(* Schneider Machine Expert - Basic project 152024, file version 2.7.0.0 *)
(* ProjectInformations: Name=New project *)

HARDWARE
  Cpu 0: TM221CE16R
  ModuleExtensionObject 0: TM3DM24R/G
  EthernetConfiguration: NetworkName=M221, IpAllocationMode=FixedAddress, IpAddress=0.0.0.0, SubnetMask=0.0.0.0
  SerialLineConfiguration: Baud=Baud19200, Parity=ParityEven, DataBits=DataBits8, StopBits=StopBits1, PhysicalMedium=PhysicalMediumRs485, TransmissionMode=TransmissionModeModbusRtu, SlaveId=1, Addressing=SlaveAddressing
  MastTask: UsePeriodScanMode=false, PeriodScan=100
  FastTask: Period=255
  CpuBehavior: StartingMode=StartAsPreviousState, AutoSaveRamOnEeprom=true, WatchdogPeriod=250

SYMBOLS  (address, symbol, comment, settings)
  %M0       WATF4  "Was At Floor 4"
  %M1       WATF1  "Was At Floor 1"
  %M2       WATF2  "Was At Floor 2"
  %M3       WATF3  "Was At Floor 3"
  %M4       F1CALL
  %M5       F2CALL
  %M6       F3CALL
  %M7       ATF1  "At Floor 1"
  %M8       ATF2  "At Floor 2"
  %M9       ATF3  "At Floor 3"
  %M10      F4CALL
  %M11      ATF4
  %M12      DOOR_CNT
  %M30      F1LATCH
  %M31      F2LATCH
  %M32      F3LATCH
  %M35        "attaxk"
  %TM0        [Preset=5000, Base=OneMilliSeconds]
  %TM1        [Preset=1000, Base=OneMilliSeconds]
  %TM2        [Preset=30]
  %TM3        [Preset=7, Base=OneSecond]
  %I0.0     LS1
  %I0.1     LS2
  %I0.2     LS3
  %I0.3     LDR_CLOSE
  %I0.4     ECB4
  %I0.5     ECB1
  %I0.6     ECB2
  %I0.7     ECB3
  %I0.8     LDR_OPEN
  %Q0.0     UP
  %Q0.1     DOWN
  %Q0.2     FD_C
  %Q0.3     DOOR_OPEN
  %Q0.4     FD_AGD
  %Q0.5     FD_E
  %Q0.6     FD_CLOSE

POU What Floor
  (* SectionNumber=0 *)

// Rung 0
  LD %I0.0                (* LS1 *)
  S %M1                   (* WATF1 *)
  R %M2                   (* WATF2 *)
  R %M3                   (* WATF3 *)
  ST %M7                  (* ATF1 *)
  R %M0                   (* WATF4 *)
  // as ST:
  //   IF LS1 THEN WATF1 := TRUE; END_IF;
  //   IF LS1 THEN WATF2 := FALSE; END_IF;
  //   IF LS1 THEN WATF3 := FALSE; END_IF;
  //   ATF1 := LS1;
  //   IF LS1 THEN WATF4 := FALSE; END_IF;

// Rung 1
  LD %I0.1                (* LS2 *)
  R %M1                   (* WATF1 *)
  S %M2                   (* WATF2 *)
  R %M3                   (* WATF3 *)
  ST %M8                  (* ATF2 *)
  R %M0                   (* WATF4 *)
  // as ST:
  //   IF LS2 THEN WATF1 := FALSE; END_IF;
  //   IF LS2 THEN WATF2 := TRUE; END_IF;
  //   IF LS2 THEN WATF3 := FALSE; END_IF;
  //   ATF2 := LS2;
  //   IF LS2 THEN WATF4 := FALSE; END_IF;

// Rung 2
  LD %I0.2                (* LS3 *)
  R %M1                   (* WATF1 *)
  R %M2                   (* WATF2 *)
  S %M3                   (* WATF3 *)
  ST %M9                  (* ATF3 *)
  R %M0                   (* WATF4 *)
  // as ST:
  //   IF LS3 THEN WATF1 := FALSE; END_IF;
  //   IF LS3 THEN WATF2 := FALSE; END_IF;
  //   IF LS3 THEN WATF3 := TRUE; END_IF;
  //   ATF3 := LS3;
  //   IF LS3 THEN WATF4 := FALSE; END_IF;

POU First Called
  (* SectionNumber=0 *)

// Rung 3
  LD %I0.5                (* ECB1 *)
  ANDN %M7                (* ATF1 *)
  S %M4                   (* F1CALL *)
  // as ST:
  //   IF ECB1 AND NOT ATF1 THEN F1CALL := TRUE; END_IF;

// Rung 4
  LD %M4                  (* F1CALL *)
  S %Q0.1                 (* DOWN *)
  // as ST:
  //   IF F1CALL THEN DOWN := TRUE; END_IF;

// Rung 5
  LD %M7                  (* ATF1 *)
  AND %M4                 (* F1CALL *)
  R %Q0.1                 (* DOWN *)
  // as ST:
  //   IF ATF1 AND F1CALL THEN DOWN := FALSE; END_IF;

// Rung 6
  LD %M7                  (* ATF1 *)
  R %M4                   (* F1CALL *)
  // as ST:
  //   IF ATF1 THEN F1CALL := FALSE; END_IF;

POU Second Called
  (* SectionNumber=0 *)

// Rung 7
  LD %I0.6                (* ECB2 *)
  ANDN %M8                (* ATF2 *)
  S %M5                   (* F2CALL *)
  // as ST:
  //   IF ECB2 AND NOT ATF2 THEN F2CALL := TRUE; END_IF;

// Rung 8
  LD %M5                  (* F2CALL *)
  AND %M1                 (* WATF1 *)
  S %Q0.0                 (* UP *)
  // as ST:
  //   IF F2CALL AND WATF1 THEN UP := TRUE; END_IF;

// Rung 9
  LD %M5                  (* F2CALL *)
  AND( %M3                (* WATF3 *)
  OR %M0                  (* WATF4 *)
  )
  S %Q0.1                 (* DOWN *)
  // as ST:
  //   IF F2CALL AND (WATF3 OR WATF4) THEN DOWN := TRUE; END_IF;

// Rung 10
  LD %M8                  (* ATF2 *)
  AND %M5                 (* F2CALL *)
  R %Q0.0                 (* UP *)
  R %Q0.1                 (* DOWN *)
  // as ST:
  //   IF ATF2 AND F2CALL THEN UP := FALSE; END_IF;
  //   IF ATF2 AND F2CALL THEN DOWN := FALSE; END_IF;

// Rung 11
  LD %M8                  (* ATF2 *)
  R %M5                   (* F2CALL *)
  // as ST:
  //   IF ATF2 THEN F2CALL := FALSE; END_IF;

POU Third Called
  (* SectionNumber=0 *)

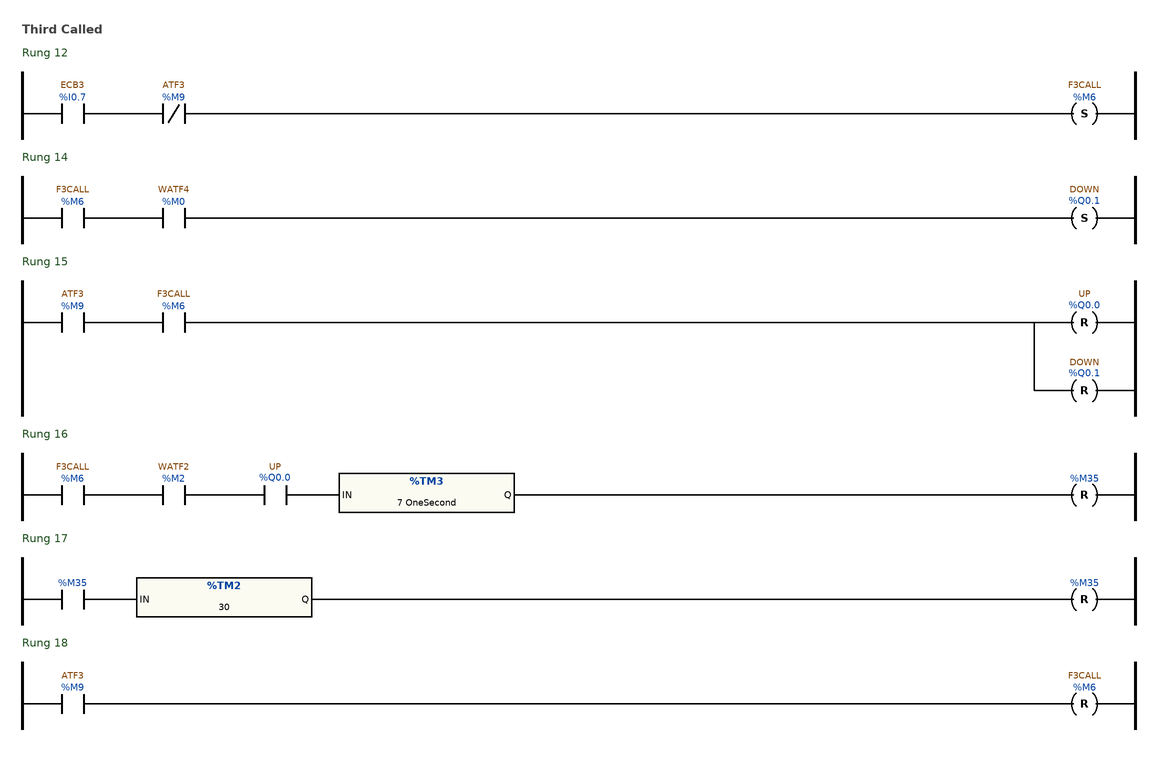

// Rung 12
  LD %I0.7                (* ECB3 *)
  ANDN %M9                (* ATF3 *)
  S %M6                   (* F3CALL *)
  // as ST:
  //   IF ECB3 AND NOT ATF3 THEN F3CALL := TRUE; END_IF;

// Rung 13
  LD %M6                  (* F3CALL *)
  AND( %M2                (* WATF2 *)
  OR %M1                  (* WATF1 *)
  )
  ANDN %M35
  S %Q0.0                 (* UP *)
  AND %M35
  R %Q0.0                 (* UP *)
  // as ST:
  //   IF F3CALL AND (WATF2 OR WATF1) AND NOT %M35 THEN UP := TRUE; END_IF;
  //   IF F3CALL AND (WATF2 OR WATF1) AND NOT %M35 AND %M35 THEN UP := FALSE; END_IF;

// Rung 14
  LD %M6                  (* F3CALL *)
  AND %M0                 (* WATF4 *)
  S %Q0.1                 (* DOWN *)
  // as ST:
  //   IF F3CALL AND WATF4 THEN DOWN := TRUE; END_IF;

// Rung 15
  LD %M9                  (* ATF3 *)
  AND %M6                 (* F3CALL *)
  R %Q0.0                 (* UP *)
  R %Q0.1                 (* DOWN *)
  // as ST:
  //   IF ATF3 AND F3CALL THEN UP := FALSE; END_IF;
  //   IF ATF3 AND F3CALL THEN DOWN := FALSE; END_IF;

// Rung 16
  BLK %TM3
  LD %M6                  (* F3CALL *)
  AND %M2                 (* WATF2 *)
  AND %Q0.0               (* UP *)
  IN
  OUT_BLK
  LD Q
  R %M35
  END_BLK
  // as ST:
  //   %TM3(IN := F3CALL AND WATF2 AND UP);
  //   IF %TM3.Q THEN %M35 := FALSE; END_IF;

// Rung 17
  BLK %TM2
  LD %M35
  IN
  OUT_BLK
  LD Q
  R %M35
  END_BLK
  // as ST:
  //   %TM2(IN := %M35);
  //   IF %TM2.Q THEN %M35 := FALSE; END_IF;

// Rung 18
  LD %M9                  (* ATF3 *)
  R %M6                   (* F3CALL *)
  // as ST:
  //   IF ATF3 THEN F3CALL := FALSE; END_IF;

POU Floor Display
  (* SectionNumber=0 *)

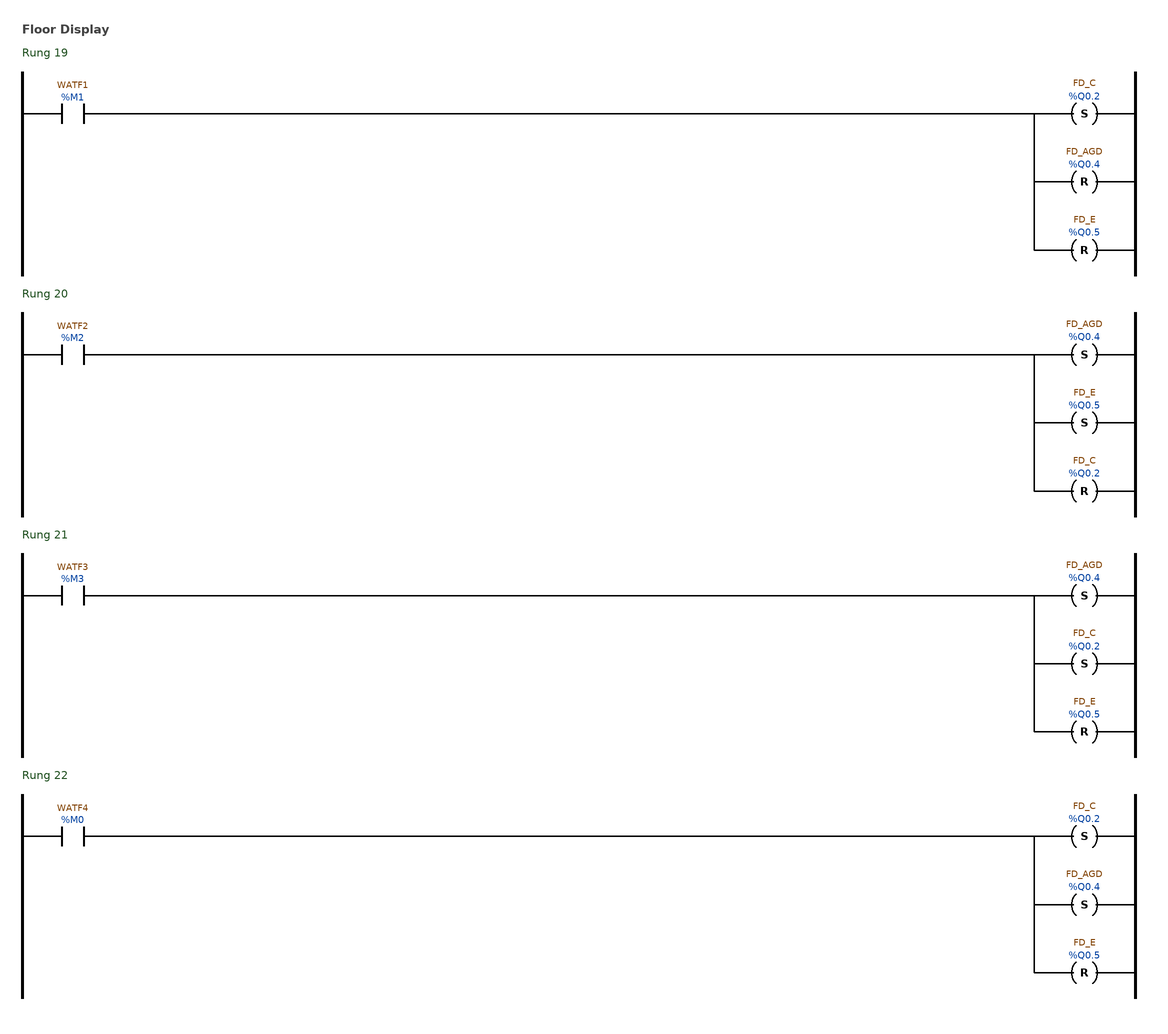

// Rung 19
  LD %M1                  (* WATF1 *)
  S %Q0.2                 (* FD_C *)
  R %Q0.4                 (* FD_AGD *)
  R %Q0.5                 (* FD_E *)
  // as ST:
  //   IF WATF1 THEN FD_C := TRUE; END_IF;
  //   IF WATF1 THEN FD_AGD := FALSE; END_IF;
  //   IF WATF1 THEN FD_E := FALSE; END_IF;

// Rung 20
  LD %M2                  (* WATF2 *)
  S %Q0.4                 (* FD_AGD *)
  S %Q0.5                 (* FD_E *)
  R %Q0.2                 (* FD_C *)
  // as ST:
  //   IF WATF2 THEN FD_AGD := TRUE; END_IF;
  //   IF WATF2 THEN FD_E := TRUE; END_IF;
  //   IF WATF2 THEN FD_C := FALSE; END_IF;

// Rung 21
  LD %M3                  (* WATF3 *)
  S %Q0.4                 (* FD_AGD *)
  S %Q0.2                 (* FD_C *)
  R %Q0.5                 (* FD_E *)
  // as ST:
  //   IF WATF3 THEN FD_AGD := TRUE; END_IF;
  //   IF WATF3 THEN FD_C := TRUE; END_IF;
  //   IF WATF3 THEN FD_E := FALSE; END_IF;

// Rung 22
  LD %M0                  (* WATF4 *)
  S %Q0.2                 (* FD_C *)
  S %Q0.4                 (* FD_AGD *)
  R %Q0.5                 (* FD_E *)
  // as ST:
  //   IF WATF4 THEN FD_C := TRUE; END_IF;
  //   IF WATF4 THEN FD_AGD := TRUE; END_IF;
  //   IF WATF4 THEN FD_E := FALSE; END_IF;

POU Elevator Door
  (* SectionNumber=0 *)

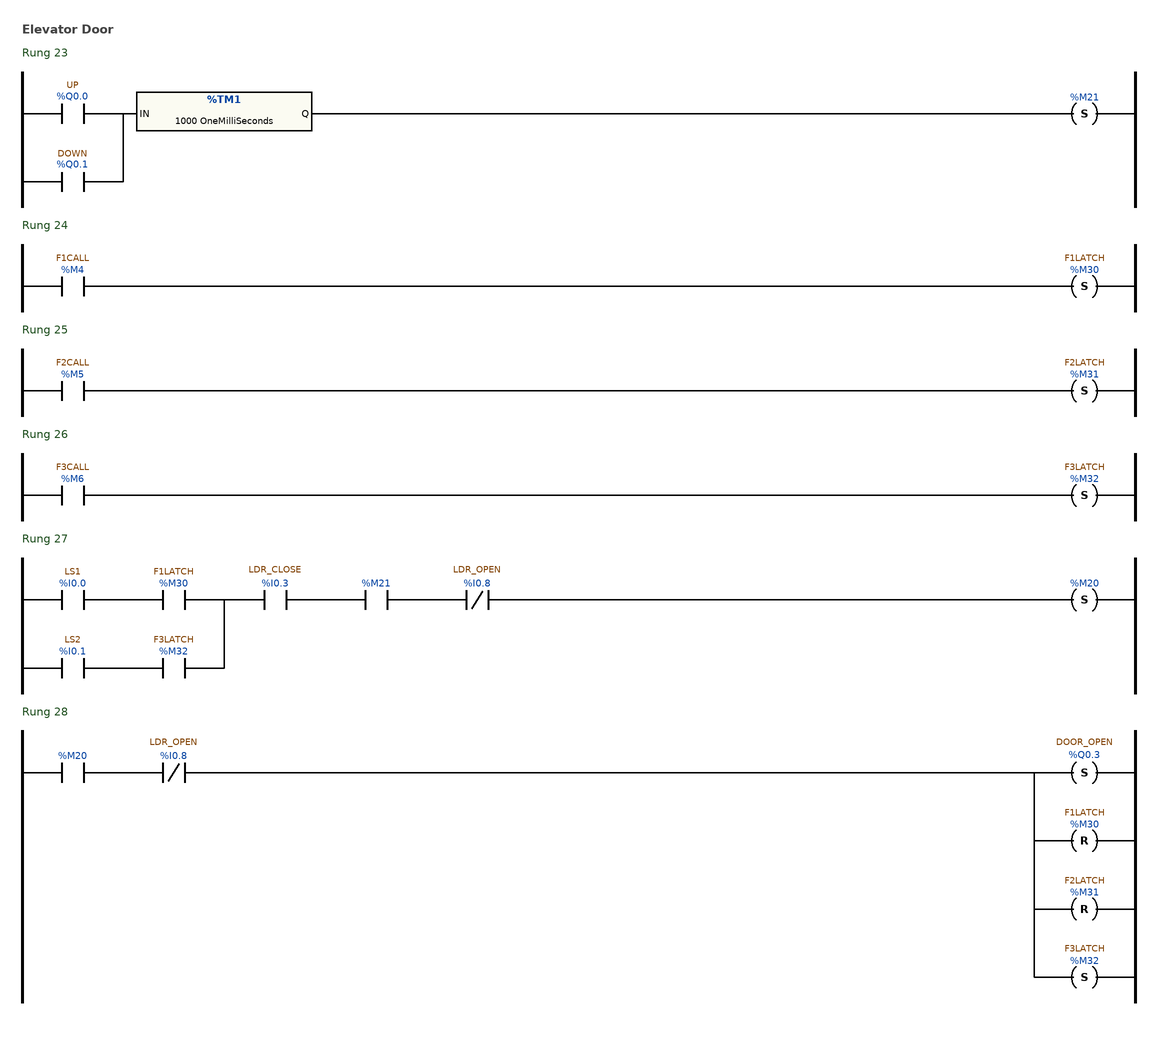

// Rung 23
  BLK %TM1
  LD %Q0.0                (* UP *)
  OR %Q0.1                (* DOWN *)
  IN
  OUT_BLK
  LD Q
  S %M21
  END_BLK
  // as ST:
  //   %TM1(IN := UP OR DOWN);
  //   IF %TM1.Q THEN %M21 := TRUE; END_IF;

// Rung 24
  LD %M4                  (* F1CALL *)
  S %M30                  (* F1LATCH *)
  // as ST:
  //   IF F1CALL THEN F1LATCH := TRUE; END_IF;

// Rung 25
  LD %M5                  (* F2CALL *)
  S %M31                  (* F2LATCH *)
  // as ST:
  //   IF F2CALL THEN F2LATCH := TRUE; END_IF;

// Rung 26
  LD %M6                  (* F3CALL *)
  S %M32                  (* F3LATCH *)
  // as ST:
  //   IF F3CALL THEN F3LATCH := TRUE; END_IF;

// Rung 27
  LD %I0.0                (* LS1 *)
  AND %M30                (* F1LATCH *)
  OR( %I0.1               (* LS2 *)
  AND %M32                (* F3LATCH *)
  )
  AND %I0.3               (* LDR_CLOSE *)
  AND %M21
  ANDN %I0.8              (* LDR_OPEN *)
  S %M20
  // as ST:
  //   IF (LS1 AND F1LATCH OR LS2 AND F3LATCH) AND LDR_CLOSE AND %M21 AND NOT LDR_OPEN THEN %M20 := TRUE; END_IF;

// Rung 28
  LD %M20
  ANDN %I0.8              (* LDR_OPEN *)
  S %Q0.3                 (* DOOR_OPEN *)
  R %M30                  (* F1LATCH *)
  R %M31                  (* F2LATCH *)
  S %M32                  (* F3LATCH *)
  // as ST:
  //   IF %M20 AND NOT LDR_OPEN THEN DOOR_OPEN := TRUE; END_IF;
  //   IF %M20 AND NOT LDR_OPEN THEN F1LATCH := FALSE; END_IF;
  //   IF %M20 AND NOT LDR_OPEN THEN F2LATCH := FALSE; END_IF;
  //   IF %M20 AND NOT LDR_OPEN THEN F3LATCH := TRUE; END_IF;

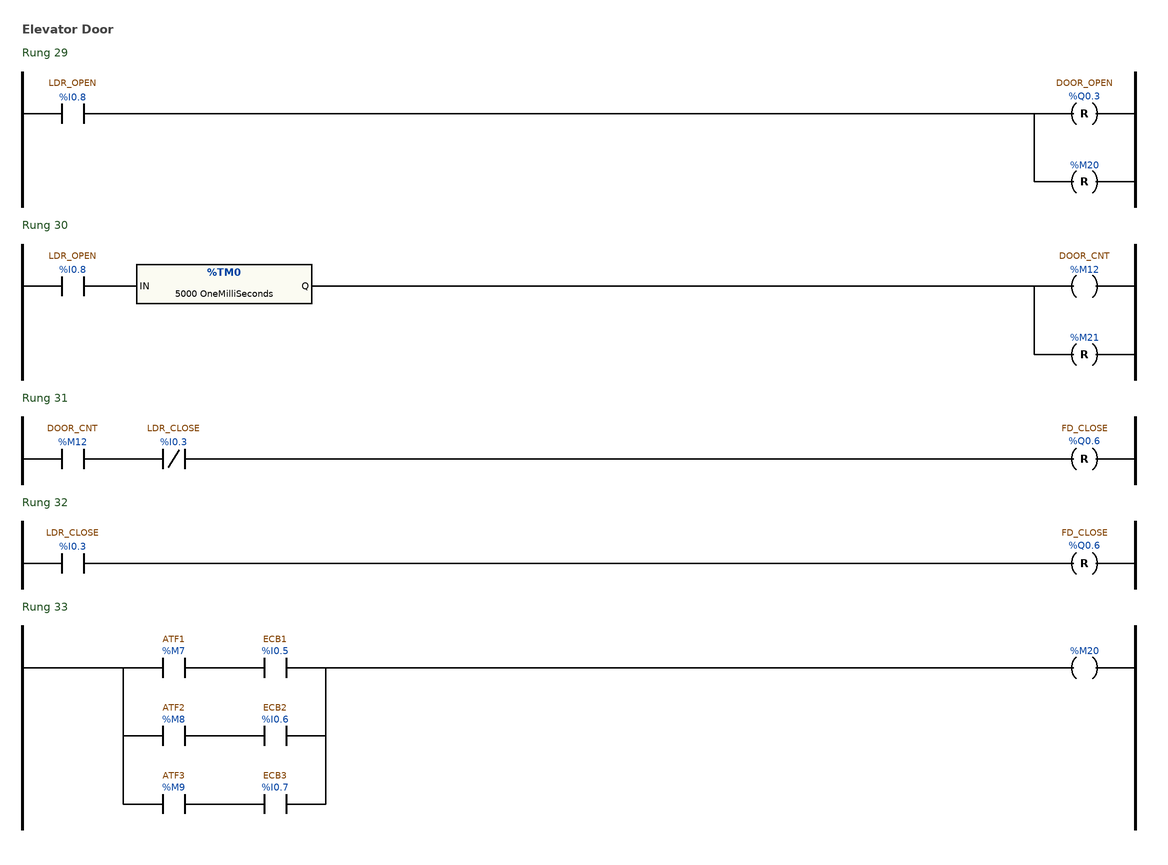

// Rung 29
  LD %I0.8                (* LDR_OPEN *)
  R %Q0.3                 (* DOOR_OPEN *)
  R %M20
  // as ST:
  //   IF LDR_OPEN THEN DOOR_OPEN := FALSE; END_IF;
  //   IF LDR_OPEN THEN %M20 := FALSE; END_IF;

// Rung 30
  BLK %TM0
  LD %I0.8                (* LDR_OPEN *)
  IN
  OUT_BLK
  LD Q
  ST %M12                 (* DOOR_CNT *)
  R %M21
  END_BLK
  // as ST:
  //   %TM0(IN := LDR_OPEN);
  //   DOOR_CNT := %TM0.Q;
  //   IF %TM0.Q THEN %M21 := FALSE; END_IF;

// Rung 31
  LD %M12                 (* DOOR_CNT *)
  ANDN %I0.3              (* LDR_CLOSE *)
  R %Q0.6                 (* FD_CLOSE *)
  // as ST:
  //   IF DOOR_CNT AND NOT LDR_CLOSE THEN FD_CLOSE := FALSE; END_IF;

// Rung 32
  LD %I0.3                (* LDR_CLOSE *)
  R %Q0.6                 (* FD_CLOSE *)
  // as ST:
  //   IF LDR_CLOSE THEN FD_CLOSE := FALSE; END_IF;

// Rung 33
  LD 1
  AND( %M7                (* ATF1 *)
  AND %I0.5               (* ECB1 *)
  OR( %M8                 (* ATF2 *)
  AND %I0.6               (* ECB2 *)
  )
  OR( %M9                 (* ATF3 *)
  AND %I0.7               (* ECB3 *)
  )
  )
  ST %M20
  // as ST:
  //   %M20 := ATF1 AND ECB1 OR ATF2 AND ECB2 OR ATF3 AND ECB3;
